(*
Casts I_Component to I_Tag
*)
FUNCTION ICompToITag : Result
VAR_INPUT
	iSource	: I_Component;
END_VAR
VAR_OUTPUT
	iDest	: I_Tag;
END_VAR

IF iSource = 0 THEN
	ICompToITag := Err.Itf0;
	RETURN;
END_IF

IF __QUERYINTERFACE(iSource, iDest) THEN
	ICompToITag := Ok;
ELSE
	iDest := 0;
	ICompToITag := Err.NoMatch;
END_IF

END_FUNCTION

(* stored: Version 1.1.0.1
   POU ICompToITag: Id {3feb1b07-c695-429c-b10c-285305651b80}, SpecialFunc None *)
